(* CODESYS project 1102_xlh_stamp_rover_ddsm210_imu_client.project
   Author: 3S - Smart Software Solutions GmbH
   Version: 1.0.0.0
   Description: Receives some incoming messages and echoes them with CAN-ID +1
   Title: CAN Bus API Example
   Company: 3S - Smart Software Solutions GmbH

Project tree, tasks and I/O mapping:
  xLH_base : CODESYS Control for Raspberry Pi 64 SL, CODESYS, order no. 2302000009, version 4.20.0.0
    application app
      libraries: Standard, 3.5.22.0 (System); Util, 3.5.22.0 (System); VisuDialogs, * (System); Memory, * (3S - Smart Software Solutions GmbH); CmpBitmapPool, * (System); CAN API, 1.0.0.4 (CODESYS)
      task MAIN_TASK (cyclic, interval 5 ms, priority 0) calls MAIN
      program MAIN [ST]
    SoftMotion General Axis Pool
    GPIOs_A_B : GPIOs B+/Pi2, CODESYS, version 4.20.0.0
        unmapped channels: digital inputs (GPIO0..GPIO31), digital outputs (GPIO0..GPIO31)
    Onewire
    Camera device
      <Leer>
    SPI
    I²C
    CANbus : CANbus, CODESYS, version 4.3.0.0
        settings: Baudrate = 1000 kbit/s
      xlh_ddsm210_ultrasonic : CANopen Device, CODESYS, version 4.3.0.0
          settings: Vendor Name = 'xemax ag'; Product Name = 'xlh_ddsm210_imu'; OD_ObjectCount = 16#001D; Objects.Objects = (wIndex := 16#1000, bySubCnt := 16#1); Objects.Objects = (wIndex := 16#1001, bySubCnt := 16#1); Objects.Objects = (wIndex := 16#1003, bySubCnt := 16#04); Objects.Objects = (wIndex := 16#1005, bySubCnt := 16#1); Objects.Objects = (wIndex := 16#1006, bySubCnt := 16#1); Objects.Objects = (wIndex := 16#100C, bySubCnt := 16#1); Objects.Objects = (wIndex := 16#100D, bySubCnt := 16#1); Objects.Objects = (wIndex := 16#1016, bySubCnt := 16#02); Objects.Objects = (wIndex := 16#1018, bySubCnt := 16#04); Objects.Objects = (wIndex := 16#1200, bySubCnt := 16#03); Objects.Objects = (wIndex := 16#1400, bySubCnt := 16#03); Objects.Objects = (wIndex := 16#1600, bySubCnt := 16#05); Objects.Objects = (wIndex := 16#1800, bySubCnt := 16#06); Objects.Objects = (wIndex := 16#1801, bySubCnt := 16#06); Objects.Objects = (wIndex := 16#1802, bySubCnt := 16#06); Objects.Objects = (wIndex := 16#1A00, bySubCnt := 16#05); Objects.Objects = (wIndex := 16#1A01, bySubCnt := 16#03); Objects.Objects = (wIndex := 16#1A02, bySubCnt := 16#04); Objects.Objects = (wIndex := 16#3000, bySubCnt := 16#02); Objects.Objects = (wIndex := 16#3001, bySubCnt := 16#02); Objects.Objects = (wIndex := 16#3002, bySubCnt := 16#02); Objects.Objects = (wIndex := 16#3003, bySubCnt := 16#02); Objects.Objects = (wIndex := 16#3800, bySubCnt := 16#02); Objects.Objects = (wIndex := 16#3801, bySubCnt := 16#02); Objects.Objects = (wIndex := 16#3802, bySubCnt := 16#02); Objects.Objects = (wIndex := 16#3803, bySubCnt := 16#02); Objects.Objects = (wIndex := 16#3804, bySubCnt := 16#02); Objects.Objects = (wIndex := 16#3805, bySubCnt := 16#02); Objects.Objects = (wIndex := 16#3806, bySubCnt := 16#04); SubObjects.SubObjects = (eObjProperties := 16#0001, eDataType := 16#07, udiSize := 16#00000004, xwData := 0, xwDefault := 0, bySubIdx := 16#00); SubObjects.SubObjects = (eObjProperties := 16#0001, eDataType := 16#05, udiSize := 16#00000001, xwData := 0, xwDefault := 0, bySubIdx := 16#00); SubObjects.SubObjects = (eObjProperties := 16#0003, eDataType := 16#05, udiSize := 16#00000001, xwData := 0, xwDefault := 0, bySubIdx := 16#00); SubObjects.SubObjects = (eObjProperties := 16#0001, eDataType := 16#07, udiSize := 16#00000004, xwData := 0, xwDefault := 0, bySubIdx := 16#01); SubObjects.SubObjects = (eObjProperties := 16#0001, eDataType := 16#07, udiSize := 16#00000004, xwData := 0, xwDefault := 0, bySubIdx := 16#02); SubObjects.SubObjects = (eObjProperties := 16#0001, eDataType := 16#07, udiSize := 16#00000004, xwData := 0, xwDefault := 0, bySubIdx := 16#03); SubObjects.SubObjects = (eObjProperties := 16#0003, eDataType := 16#07, udiSize := 16#00000004, xwData := 0, xwDefault := 0, bySubIdx := 16#00); SubObjects.SubObjects = (eObjProperties := 16#0003, eDataType := 16#05, udiSize := 16#00000001, xwData := 0, xwDefault := 3, bySubIdx := 16#00);
            SubObjects.SubObjects = (eObjProperties := 16#0001, eDataType := 16#05, udiSize := 16#00000001, xwData := 0, xwDefault := 1, bySubIdx := 16#00); SubObjects.SubObjects = (eObjProperties := 16#0003, eDataType := 16#07, udiSize := 16#00000004, xwData := 0, xwDefault := 0, bySubIdx := 16#01); SubObjects.SubObjects = (eObjProperties := 16#0001, eDataType := 16#05, udiSize := 16#00000001, xwData := 0, xwDefault := 3, bySubIdx := 16#00); SubObjects.SubObjects = (eObjProperties := 16#0001, eDataType := 16#07, udiSize := 16#00000004, xwData := 0, xwDefault := 1, bySubIdx := 16#03); SubObjects.SubObjects = (eObjProperties := 16#0001, eDataType := 16#05, udiSize := 16#00000001, xwData := 0, xwDefault := 2, bySubIdx := 16#00); SubObjects.SubObjects = (eObjProperties := 16#0001, eDataType := 16#05, udiSize := 16#00000001, xwData := 0, xwDefault := 2, bySubIdx := 16#00); SubObjects.SubObjects = (eObjProperties := 16#0001, eDataType := 16#05, udiSize := 16#00000001, xwData := 0, xwDefault := 4, bySubIdx := 16#00); SubObjects.SubObjects = (eObjProperties := 16#0001, eDataType := 16#05, udiSize := 16#00000001, xwData := 0, xwDefault := 5, bySubIdx := 16#00); SubObjects.SubObjects = (eObjProperties := 16#0003, eDataType := 16#06, udiSize := 16#00000002, xwData := 0, xwDefault := 0, bySubIdx := 16#03); SubObjects.SubObjects = (eObjProperties := 16#0003, eDataType := 16#05, udiSize := 16#00000001, xwData := 0, xwDefault := 0, bySubIdx := 16#04); SubObjects.SubObjects = (eObjProperties := 16#0003, eDataType := 16#06, udiSize := 16#00000002, xwData := 0, xwDefault := 0, bySubIdx := 16#05); SubObjects.SubObjects = (eObjProperties := 16#0001, eDataType := 16#05, udiSize := 16#00000001, xwData := 0, xwDefault := 5, bySubIdx := 16#00); SubObjects.SubObjects = (eObjProperties := 16#0003, eDataType := 16#06, udiSize := 16#00000002, xwData := 0, xwDefault := 0, bySubIdx := 16#03); SubObjects.SubObjects = (eObjProperties := 16#0003, eDataType := 16#05, udiSize := 16#00000001, xwData := 0, xwDefault := 0, bySubIdx := 16#04); SubObjects.SubObjects = (eObjProperties := 16#0003, eDataType := 16#06, udiSize := 16#00000002, xwData := 0, xwDefault := 0, bySubIdx := 16#05); SubObjects.SubObjects = (eObjProperties := 16#0001, eDataType := 16#05, udiSize := 16#00000001, xwData := 0, xwDefault := 5, bySubIdx := 16#00); SubObjects.SubObjects = (eObjProperties := 16#0003, eDataType := 16#06, udiSize := 16#00000002, xwData := 0, xwDefault := 0, bySubIdx := 16#03); SubObjects.SubObjects = (eObjProperties := 16#0003, eDataType := 16#05, udiSize := 16#00000001, xwData := 0, xwDefault := 0, bySubIdx := 16#04); SubObjects.SubObjects = (eObjProperties := 16#0003, eDataType := 16#06, udiSize := 16#00000002, xwData := 0, xwDefault := 0, bySubIdx := 16#05); SubObjects.SubObjects = (eObjProperties := 16#0001, eDataType := 16#05, udiSize := 16#00000001, xwData := 0, xwDefault := 4, bySubIdx := 16#00); SubObjects.SubObjects = (eObjProperties := 16#0001, eDataType := 16#05, udiSize := 16#00000001, xwData := 0, xwDefault := 2, bySubIdx := 16#00); SubObjects.SubObjects = (eObjProperties := 16#0001, eDataType := 16#05, udiSize := 16#00000001, xwData := 0, xwDefault := 3, bySubIdx := 16#00); SubObjects.SubObjects = (eObjProperties := 16#0001, eDataType := 16#05, udiSize := 16#00000001, xwData := 0, xwDefault := 1, bySubIdx := 16#00); SubObjects.SubObjects = (eObjProperties := 16#0003, eDataType := 16#03, udiSize := 16#00000002, xwData := 0, xwDefault := 0, bySubIdx := 16#01); SubObjects.SubObjects = (eObjProperties := 16#0001, eDataType := 16#05, udiSize := 16#00000001, xwData := 0, xwDefault := 1, bySubIdx := 16#00); SubObjects.SubObjects = (eObjProperties := 16#0003, eDataType := 16#05, udiSize := 16#00000001, xwData := 0, xwDefault := 0, bySubIdx := 16#01); SubObjects.SubObjects = (eObjProperties := 16#0001, eDataType := 16#05, udiSize := 16#00000001, xwData := 0, xwDefault := 1, bySubIdx := 16#00); SubObjects.SubObjects = (eObjProperties := 16#0003, eDataType := 16#03, udiSize := 16#00000002, xwData := 0, xwDefault := 0, bySubIdx := 16#01); SubObjects.SubObjects = (eObjProperties := 16#0001, eDataType := 16#05, udiSize := 16#00000001, xwData := 0, xwDefault := 1, bySubIdx := 16#00); SubObjects.SubObjects = (eObjProperties := 16#0003, eDataType := 16#05, udiSize := 16#00000001, xwData := 0, xwDefault := 0, bySubIdx := 16#01); SubObjects.SubObjects = (eObjProperties := 16#0001, eDataType := 16#05, udiSize := 16#00000001, xwData := 0, xwDefault := 1, bySubIdx := 16#00); SubObjects.SubObjects = (eObjProperties := 16#0001, eDataType := 16#03, udiSize := 16#00000002, xwData := 0, xwDefault := 0, bySubIdx := 16#01); SubObjects.SubObjects = (eObjProperties := 16#0001, eDataType := 16#05, udiSize := 16#00000001, xwData := 0, xwDefault := 1, bySubIdx := 16#00); SubObjects.SubObjects = (eObjProperties := 16#0001, eDataType := 16#03, udiSize := 16#00000002, xwData := 0, xwDefault := 0, bySubIdx := 16#01); SubObjects.SubObjects = (eObjProperties := 16#0001, eDataType := 16#05, udiSize := 16#00000001, xwData := 0, xwDefault := 1, bySubIdx := 16#00); SubObjects.SubObjects = (eObjProperties := 16#0001, eDataType := 16#05, udiSize := 16#00000001, xwData := 0, xwDefault := 0, bySubIdx := 16#01); SubObjects.SubObjects = (eObjProperties := 16#0001, eDataType := 16#05, udiSize := 16#00000001, xwData := 0, xwDefault := 1, bySubIdx := 16#00); SubObjects.SubObjects = (eObjProperties := 16#0001, eDataType := 16#05, udiSize := 16#00000001, xwData := 0, xwDefault := 0, bySubIdx := 16#01); SubObjects.SubObjects = (eObjProperties := 16#0001, eDataType := 16#05, udiSize := 16#00000001, xwData := 0, xwDefault := 1, bySubIdx := 16#00); SubObjects.SubObjects = (eObjProperties := 16#0001, eDataType := 16#04, udiSize := 16#00000004, xwData := 0, xwDefault := 0, bySubIdx := 16#01);
            SubObjects.SubObjects = (eObjProperties := 16#0001, eDataType := 16#05, udiSize := 16#00000001, xwData := 0, xwDefault := 1, bySubIdx := 16#00); SubObjects.SubObjects = (eObjProperties := 16#0001, eDataType := 16#06, udiSize := 16#00000002, xwData := 0, xwDefault := 0, bySubIdx := 16#01); SubObjects.SubObjects = (eObjProperties := 16#0001, eDataType := 16#05, udiSize := 16#00000001, xwData := 0, xwDefault := 3, bySubIdx := 16#00); SubObjects.SubObjects = (eObjProperties := 16#0001, eDataType := 16#03, udiSize := 16#00000002, xwData := 0, xwDefault := 0, bySubIdx := 16#01); SubObjects.SubObjects = (eObjProperties := 16#0001, eDataType := 16#03, udiSize := 16#00000002, xwData := 0, xwDefault := 0, bySubIdx := 16#02); SubObjects.SubObjects = (eObjProperties := 16#0001, eDataType := 16#03, udiSize := 16#00000002, xwData := 0, xwDefault := 0, bySubIdx := 16#03); ObjectsOfflineInfo.Predefined Error Field.Index = 16#00001003; ObjectsOfflineInfo.Predefined Error Field.ObjectOwner = 16#00; ObjectsOfflineInfo.Predefined Error Field.ObjectType = 16#00000008; ObjectsOfflineInfo.Predefined Error Field.ObjectFlags = 16#00000000; ObjectsOfflineInfo.Consumer Heartbeat Time.Index = 16#00001016; ObjectsOfflineInfo.Consumer Heartbeat Time.ObjectOwner = 16#00; ObjectsOfflineInfo.Consumer Heartbeat Time.ObjectType = 16#00000008; ObjectsOfflineInfo.Consumer Heartbeat Time.ObjectFlags = 16#00000000; ObjectsOfflineInfo.Identity Object.Index = 16#00001018; ObjectsOfflineInfo.Identity Object.ObjectOwner = 16#00; ObjectsOfflineInfo.Identity Object.ObjectType = 16#00000009; ObjectsOfflineInfo.Identity Object.ObjectFlags = 16#00000000; ObjectsOfflineInfo.ServerSdoParameter.Index = 16#00001200; ObjectsOfflineInfo.ServerSdoParameter.ObjectOwner = 16#00; ObjectsOfflineInfo.ServerSdoParameter.ObjectType = 16#00000009; ObjectsOfflineInfo.ServerSdoParameter.ObjectFlags = 16#00000000; ObjectsOfflineInfo.RPDO communication parameter.Index = 16#00001400; ObjectsOfflineInfo.RPDO communication parameter.ObjectOwner = 16#03; ObjectsOfflineInfo.RPDO communication parameter.ObjectType = 16#00000009; ObjectsOfflineInfo.RPDO communication parameter.ObjectFlags = 16#00000000; ObjectsOfflineInfo.RPDO mapping parameter.Index = 16#00001600; ObjectsOfflineInfo.RPDO mapping parameter.ObjectOwner = 16#03; ObjectsOfflineInfo.RPDO mapping parameter.ObjectType = 16#00000009; ObjectsOfflineInfo.RPDO mapping parameter.ObjectFlags = 16#00000000; ObjectsOfflineInfo.TPDO communication parameter.Index = 16#00001800; ObjectsOfflineInfo.TPDO communication parameter.ObjectOwner = 16#03; ObjectsOfflineInfo.TPDO communication parameter.ObjectType = 16#00000009; ObjectsOfflineInfo.TPDO communication parameter.ObjectFlags = 16#00000000; ObjectsOfflineInfo.TPDO communication parameter.Index = 16#00001801; ObjectsOfflineInfo.TPDO communication parameter.ObjectOwner = 16#03; ObjectsOfflineInfo.TPDO communication parameter.ObjectType = 16#00000009; ObjectsOfflineInfo.TPDO communication parameter.ObjectFlags = 16#00000000; ObjectsOfflineInfo.TPDO communication parameter.Index = 16#00001802; ObjectsOfflineInfo.TPDO communication parameter.ObjectOwner = 16#03;
            ObjectsOfflineInfo.TPDO communication parameter.ObjectType = 16#00000009; ObjectsOfflineInfo.TPDO communication parameter.ObjectFlags = 16#00000000; ObjectsOfflineInfo.TPDO mapping parameter.Index = 16#00001A00; ObjectsOfflineInfo.TPDO mapping parameter.ObjectOwner = 16#03; ObjectsOfflineInfo.TPDO mapping parameter.ObjectType = 16#00000009; ObjectsOfflineInfo.TPDO mapping parameter.ObjectFlags = 16#00000000; ObjectsOfflineInfo.TPDO mapping parameter.Index = 16#00001A01; ObjectsOfflineInfo.TPDO mapping parameter.ObjectOwner = 16#03; ObjectsOfflineInfo.TPDO mapping parameter.ObjectType = 16#00000009; ObjectsOfflineInfo.TPDO mapping parameter.ObjectFlags = 16#00000000; ObjectsOfflineInfo.TPDO mapping parameter.Index = 16#00001A02; ObjectsOfflineInfo.TPDO mapping parameter.ObjectOwner = 16#03; ObjectsOfflineInfo.TPDO mapping parameter.ObjectType = 16#00000009; ObjectsOfflineInfo.TPDO mapping parameter.ObjectFlags = 16#00000000; ObjectsOfflineInfo.set_speed.Index = 16#00003000; ObjectsOfflineInfo.set_speed.ObjectOwner = 16#03; ObjectsOfflineInfo.set_speed.ObjectType = 16#00000008; ObjectsOfflineInfo.set_speed.ObjectFlags = 16#00000000; ObjectsOfflineInfo.set_acc_time.Index = 16#00003001; ObjectsOfflineInfo.set_acc_time.ObjectOwner = 16#03; ObjectsOfflineInfo.set_acc_time.ObjectType = 16#00000008; ObjectsOfflineInfo.set_acc_time.ObjectFlags = 16#00000000; ObjectsOfflineInfo.set_current_limit.Index = 16#00003002; ObjectsOfflineInfo.set_current_limit.ObjectOwner = 16#03; ObjectsOfflineInfo.set_current_limit.ObjectType = 16#00000008; ObjectsOfflineInfo.set_current_limit.ObjectFlags = 16#00000000; ObjectsOfflineInfo.set_cmd.Index = 16#00003003; ObjectsOfflineInfo.set_cmd.ObjectOwner = 16#03; ObjectsOfflineInfo.set_cmd.ObjectType = 16#00000008; ObjectsOfflineInfo.set_cmd.ObjectFlags = 16#00000000; ObjectsOfflineInfo.speed.Index = 16#00003800; ObjectsOfflineInfo.speed.ObjectOwner = 16#03; ObjectsOfflineInfo.speed.ObjectType = 16#00000008; ObjectsOfflineInfo.speed.ObjectFlags = 16#00000000; ObjectsOfflineInfo.current.Index = 16#00003801; ObjectsOfflineInfo.current.ObjectOwner = 16#03; ObjectsOfflineInfo.current.ObjectType = 16#00000008; ObjectsOfflineInfo.current.ObjectFlags = 16#00000000; ObjectsOfflineInfo.acc_time.Index = 16#00003802; ObjectsOfflineInfo.acc_time.ObjectOwner = 16#03;
            ObjectsOfflineInfo.acc_time.ObjectType = 16#00000008; ObjectsOfflineInfo.acc_time.ObjectFlags = 16#00000000; ObjectsOfflineInfo.temperature.Index = 16#00003803; ObjectsOfflineInfo.temperature.ObjectOwner = 16#03; ObjectsOfflineInfo.temperature.ObjectType = 16#00000008; ObjectsOfflineInfo.temperature.ObjectFlags = 16#00000000; ObjectsOfflineInfo.position.Index = 16#00003804; ObjectsOfflineInfo.position.ObjectOwner = 16#03; ObjectsOfflineInfo.position.ObjectType = 16#00000008; ObjectsOfflineInfo.position.ObjectFlags = 16#00000000; ObjectsOfflineInfo.error_code.Index = 16#00003805; ObjectsOfflineInfo.error_code.ObjectOwner = 16#03; ObjectsOfflineInfo.error_code.ObjectType = 16#00000008; ObjectsOfflineInfo.error_code.ObjectFlags = 16#00000000; ObjectsOfflineInfo.imu.Index = 16#00003806; ObjectsOfflineInfo.imu.ObjectOwner = 16#03; ObjectsOfflineInfo.imu.ObjectType = 16#00000008; ObjectsOfflineInfo.imu.ObjectFlags = 16#00000000; SubObjectsOfflineInfo.Device Type.Index = 16#00001000; SubObjectsOfflineInfo.Device Type.SubIndex = 16#00; SubObjectsOfflineInfo.Device Type.PDOMapping = FALSE; SubObjectsOfflineInfo.Device Type.ObjectOwner = 16#00; SubObjectsOfflineInfo.Device Type.ObjectType = 16#00000007; SubObjectsOfflineInfo.Device Type.MinValue = ''; SubObjectsOfflineInfo.Device Type.MaxValue = ''; SubObjectsOfflineInfo.Device Type.AccessType = 'ro'; SubObjectsOfflineInfo.Device Type.IEC Variable = ''; SubObjectsOfflineInfo.Device Type.DefaultValue = '0x0'; SubObjectsOfflineInfo.Device Type.ObjectFlags = 16#00000000; SubObjectsOfflineInfo.Error Register.Index = 16#00001001; SubObjectsOfflineInfo.Error Register.SubIndex = 16#00; SubObjectsOfflineInfo.Error Register.PDOMapping = FALSE; SubObjectsOfflineInfo.Error Register.ObjectOwner = 16#00; SubObjectsOfflineInfo.Error Register.ObjectType = 16#00000007; SubObjectsOfflineInfo.Error Register.MinValue = ''; SubObjectsOfflineInfo.Error Register.MaxValue = ''; SubObjectsOfflineInfo.Error Register.AccessType = 'ro'; SubObjectsOfflineInfo.Error Register.IEC Variable = ''; SubObjectsOfflineInfo.Error Register.DefaultValue = '0x0'; SubObjectsOfflineInfo.Error Register.ObjectFlags = 16#00000000;
            SubObjectsOfflineInfo.Number of Errors.Index = 16#00001003; SubObjectsOfflineInfo.Number of Errors.SubIndex = 16#00; SubObjectsOfflineInfo.Number of Errors.PDOMapping = FALSE; SubObjectsOfflineInfo.Number of Errors.ObjectOwner = 16#00; SubObjectsOfflineInfo.Number of Errors.ObjectType = 16#00000007; SubObjectsOfflineInfo.Number of Errors.MinValue = ''; SubObjectsOfflineInfo.Number of Errors.MaxValue = ''; SubObjectsOfflineInfo.Number of Errors.AccessType = 'rw'; SubObjectsOfflineInfo.Number of Errors.IEC Variable = ''; SubObjectsOfflineInfo.Number of Errors.DefaultValue = '0'; SubObjectsOfflineInfo.Number of Errors.ObjectFlags = 16#00000000; SubObjectsOfflineInfo.Standard Error Field.Index = 16#00001003; SubObjectsOfflineInfo.Standard Error Field.SubIndex = 16#01; SubObjectsOfflineInfo.Standard Error Field.PDOMapping = FALSE; SubObjectsOfflineInfo.Standard Error Field.ObjectOwner = 16#00; SubObjectsOfflineInfo.Standard Error Field.ObjectType = 16#00000007; SubObjectsOfflineInfo.Standard Error Field.MinValue = ''; SubObjectsOfflineInfo.Standard Error Field.MaxValue = ''; SubObjectsOfflineInfo.Standard Error Field.AccessType = 'ro'; SubObjectsOfflineInfo.Standard Error Field.IEC Variable = ''; SubObjectsOfflineInfo.Standard Error Field.DefaultValue = ''; SubObjectsOfflineInfo.Standard Error Field.ObjectFlags = 16#00000000; SubObjectsOfflineInfo.Standard Error Field 2.Index = 16#00001003; SubObjectsOfflineInfo.Standard Error Field 2.SubIndex = 16#02; SubObjectsOfflineInfo.Standard Error Field 2.PDOMapping = FALSE; SubObjectsOfflineInfo.Standard Error Field 2.ObjectOwner = 16#00; SubObjectsOfflineInfo.Standard Error Field 2.ObjectType = 16#00000007; SubObjectsOfflineInfo.Standard Error Field 2.MinValue = ''; SubObjectsOfflineInfo.Standard Error Field 2.MaxValue = ''; SubObjectsOfflineInfo.Standard Error Field 2.AccessType = 'ro'; SubObjectsOfflineInfo.Standard Error Field 2.IEC Variable = ''; SubObjectsOfflineInfo.Standard Error Field 2.DefaultValue = ''; SubObjectsOfflineInfo.Standard Error Field 2.ObjectFlags = 16#00000000; SubObjectsOfflineInfo.Standard Error Field 3.Index = 16#00001003; SubObjectsOfflineInfo.Standard Error Field 3.SubIndex = 16#03; SubObjectsOfflineInfo.Standard Error Field 3.PDOMapping = FALSE; SubObjectsOfflineInfo.Standard Error Field 3.ObjectOwner = 16#00; SubObjectsOfflineInfo.Standard Error Field 3.ObjectType = 16#00000007; SubObjectsOfflineInfo.Standard Error Field 3.MinValue = ''; SubObjectsOfflineInfo.Standard Error Field 3.MaxValue = '';
            SubObjectsOfflineInfo.Standard Error Field 3.AccessType = 'ro'; SubObjectsOfflineInfo.Standard Error Field 3.IEC Variable = ''; SubObjectsOfflineInfo.Standard Error Field 3.DefaultValue = ''; SubObjectsOfflineInfo.Standard Error Field 3.ObjectFlags = 16#00000000; SubObjectsOfflineInfo.Sync COB-ID.Index = 16#00001005; SubObjectsOfflineInfo.Sync COB-ID.SubIndex = 16#00; SubObjectsOfflineInfo.Sync COB-ID.PDOMapping = FALSE; SubObjectsOfflineInfo.Sync COB-ID.ObjectOwner = 16#00; SubObjectsOfflineInfo.Sync COB-ID.ObjectType = 16#00000007; SubObjectsOfflineInfo.Sync COB-ID.MinValue = ''; SubObjectsOfflineInfo.Sync COB-ID.MaxValue = ''; SubObjectsOfflineInfo.Sync COB-ID.AccessType = 'rw'; SubObjectsOfflineInfo.Sync COB-ID.IEC Variable = ''; SubObjectsOfflineInfo.Sync COB-ID.DefaultValue = '0x80'; SubObjectsOfflineInfo.Sync COB-ID.ObjectFlags = 16#00000000; SubObjectsOfflineInfo.Communication Cycle Period.Index = 16#00001006; SubObjectsOfflineInfo.Communication Cycle Period.SubIndex = 16#00; SubObjectsOfflineInfo.Communication Cycle Period.PDOMapping = FALSE; SubObjectsOfflineInfo.Communication Cycle Period.ObjectOwner = 16#00; SubObjectsOfflineInfo.Communication Cycle Period.ObjectType = 16#00000007; SubObjectsOfflineInfo.Communication Cycle Period.MinValue = ''; SubObjectsOfflineInfo.Communication Cycle Period.MaxValue = ''; SubObjectsOfflineInfo.Communication Cycle Period.AccessType = 'rw'; SubObjectsOfflineInfo.Communication Cycle Period.IEC Variable = ''; SubObjectsOfflineInfo.Communication Cycle Period.DefaultValue = '0x0'; SubObjectsOfflineInfo.Communication Cycle Period.ObjectFlags = 16#00000000; SubObjectsOfflineInfo.Guard Time.Index = 16#0000100C; SubObjectsOfflineInfo.Guard Time.SubIndex = 16#00; SubObjectsOfflineInfo.Guard Time.PDOMapping = FALSE; SubObjectsOfflineInfo.Guard Time.ObjectOwner = 16#00; SubObjectsOfflineInfo.Guard Time.ObjectType = 16#00000007; SubObjectsOfflineInfo.Guard Time.MinValue = ''; SubObjectsOfflineInfo.Guard Time.MaxValue = ''; SubObjectsOfflineInfo.Guard Time.AccessType = 'rw'; SubObjectsOfflineInfo.Guard Time.IEC Variable = ''; SubObjectsOfflineInfo.Guard Time.DefaultValue = '200'; SubObjectsOfflineInfo.Guard Time.ObjectFlags = 16#00000000; SubObjectsOfflineInfo.Life Time Factor.Index = 16#0000100D; SubObjectsOfflineInfo.Life Time Factor.SubIndex = 16#00; SubObjectsOfflineInfo.Life Time Factor.PDOMapping = FALSE;
            SubObjectsOfflineInfo.Life Time Factor.ObjectOwner = 16#00; SubObjectsOfflineInfo.Life Time Factor.ObjectType = 16#00000007; SubObjectsOfflineInfo.Life Time Factor.MinValue = ''; SubObjectsOfflineInfo.Life Time Factor.MaxValue = ''; SubObjectsOfflineInfo.Life Time Factor.AccessType = 'rw'; SubObjectsOfflineInfo.Life Time Factor.IEC Variable = ''; SubObjectsOfflineInfo.Life Time Factor.DefaultValue = '3'; SubObjectsOfflineInfo.Life Time Factor.ObjectFlags = 16#00000000; SubObjectsOfflineInfo.Number of Entries.Index = 16#00001016; SubObjectsOfflineInfo.Number of Entries.SubIndex = 16#00; SubObjectsOfflineInfo.Number of Entries.PDOMapping = FALSE; SubObjectsOfflineInfo.Number of Entries.ObjectOwner = 16#00; SubObjectsOfflineInfo.Number of Entries.ObjectType = 16#00000007; SubObjectsOfflineInfo.Number of Entries.MinValue = ''; SubObjectsOfflineInfo.Number of Entries.MaxValue = ''; SubObjectsOfflineInfo.Number of Entries.AccessType = 'ro'; SubObjectsOfflineInfo.Number of Entries.IEC Variable = ''; SubObjectsOfflineInfo.Number of Entries.DefaultValue = '0x1'; SubObjectsOfflineInfo.Number of Entries.ObjectFlags = 16#00000000; SubObjectsOfflineInfo.Consumer Heartbeat Time.Index = 16#00001016; SubObjectsOfflineInfo.Consumer Heartbeat Time.SubIndex = 16#01; SubObjectsOfflineInfo.Consumer Heartbeat Time.PDOMapping = FALSE; SubObjectsOfflineInfo.Consumer Heartbeat Time.ObjectOwner = 16#00; SubObjectsOfflineInfo.Consumer Heartbeat Time.ObjectType = 16#00000007; SubObjectsOfflineInfo.Consumer Heartbeat Time.MinValue = ''; SubObjectsOfflineInfo.Consumer Heartbeat Time.MaxValue = ''; SubObjectsOfflineInfo.Consumer Heartbeat Time.AccessType = 'rw'; SubObjectsOfflineInfo.Consumer Heartbeat Time.IEC Variable = ''; SubObjectsOfflineInfo.Consumer Heartbeat Time.DefaultValue = '0x0'; SubObjectsOfflineInfo.Consumer Heartbeat Time.ObjectFlags = 16#00000000; SubObjectsOfflineInfo.Number of Entries.Index = 16#00001018; SubObjectsOfflineInfo.Number of Entries.SubIndex = 16#00; SubObjectsOfflineInfo.Number of Entries.PDOMapping = FALSE; SubObjectsOfflineInfo.Number of Entries.ObjectOwner = 16#00; SubObjectsOfflineInfo.Number of Entries.ObjectType = 16#00000007; SubObjectsOfflineInfo.Number of Entries.MinValue = '0x1'; SubObjectsOfflineInfo.Number of Entries.MaxValue = '0x3'; SubObjectsOfflineInfo.Number of Entries.AccessType = 'ro'; SubObjectsOfflineInfo.Number of Entries.IEC Variable = ''; SubObjectsOfflineInfo.Number of Entries.DefaultValue = '3';
            SubObjectsOfflineInfo.Number of Entries.ObjectFlags = 16#00000000; SubObjectsOfflineInfo.Vendor Id.Index = 16#00001018; SubObjectsOfflineInfo.Vendor Id.SubIndex = 16#01; SubObjectsOfflineInfo.Vendor Id.PDOMapping = FALSE; SubObjectsOfflineInfo.Vendor Id.ObjectOwner = 16#00; SubObjectsOfflineInfo.Vendor Id.ObjectType = 16#00000007; SubObjectsOfflineInfo.Vendor Id.MinValue = ''; SubObjectsOfflineInfo.Vendor Id.MaxValue = ''; SubObjectsOfflineInfo.Vendor Id.AccessType = 'ro'; SubObjectsOfflineInfo.Vendor Id.IEC Variable = ''; SubObjectsOfflineInfo.Vendor Id.DefaultValue = '801'; SubObjectsOfflineInfo.Vendor Id.ObjectFlags = 16#00000000; SubObjectsOfflineInfo.Product Code.Index = 16#00001018; SubObjectsOfflineInfo.Product Code.SubIndex = 16#02; SubObjectsOfflineInfo.Product Code.PDOMapping = FALSE; SubObjectsOfflineInfo.Product Code.ObjectOwner = 16#00; SubObjectsOfflineInfo.Product Code.ObjectType = 16#00000007; SubObjectsOfflineInfo.Product Code.MinValue = ''; SubObjectsOfflineInfo.Product Code.MaxValue = ''; SubObjectsOfflineInfo.Product Code.AccessType = 'ro'; SubObjectsOfflineInfo.Product Code.IEC Variable = ''; SubObjectsOfflineInfo.Product Code.DefaultValue = '1102'; SubObjectsOfflineInfo.Product Code.ObjectFlags = 16#00000000; SubObjectsOfflineInfo.Revision Number.Index = 16#00001018; SubObjectsOfflineInfo.Revision Number.SubIndex = 16#03; SubObjectsOfflineInfo.Revision Number.PDOMapping = FALSE; SubObjectsOfflineInfo.Revision Number.ObjectOwner = 16#00; SubObjectsOfflineInfo.Revision Number.ObjectType = 16#00000007; SubObjectsOfflineInfo.Revision Number.MinValue = ''; SubObjectsOfflineInfo.Revision Number.MaxValue = ''; SubObjectsOfflineInfo.Revision Number.AccessType = 'ro'; SubObjectsOfflineInfo.Revision Number.IEC Variable = ''; SubObjectsOfflineInfo.Revision Number.DefaultValue = '1'; SubObjectsOfflineInfo.Revision Number.ObjectFlags = 16#00000000; SubObjectsOfflineInfo.Number of Entries.Index = 16#00001200; SubObjectsOfflineInfo.Number of Entries.SubIndex = 16#00; SubObjectsOfflineInfo.Number of Entries.PDOMapping = FALSE; SubObjectsOfflineInfo.Number of Entries.ObjectOwner = 16#00; SubObjectsOfflineInfo.Number of Entries.ObjectType = 16#00000007; SubObjectsOfflineInfo.Number of Entries.MinValue = '0x2';
            SubObjectsOfflineInfo.Number of Entries.MaxValue = '0x2'; SubObjectsOfflineInfo.Number of Entries.AccessType = 'ro'; SubObjectsOfflineInfo.Number of Entries.IEC Variable = ''; SubObjectsOfflineInfo.Number of Entries.DefaultValue = '0x2'; SubObjectsOfflineInfo.Number of Entries.ObjectFlags = 16#00000000; SubObjectsOfflineInfo.COB-ID Client->Server.Index = 16#00001200; SubObjectsOfflineInfo.COB-ID Client->Server.SubIndex = 16#01; SubObjectsOfflineInfo.COB-ID Client->Server.PDOMapping = FALSE; SubObjectsOfflineInfo.COB-ID Client->Server.ObjectOwner = 16#00; SubObjectsOfflineInfo.COB-ID Client->Server.ObjectType = 16#00000007; SubObjectsOfflineInfo.COB-ID Client->Server.MinValue = ''; SubObjectsOfflineInfo.COB-ID Client->Server.MaxValue = ''; SubObjectsOfflineInfo.COB-ID Client->Server.AccessType = 'ro'; SubObjectsOfflineInfo.COB-ID Client->Server.IEC Variable = ''; SubObjectsOfflineInfo.COB-ID Client->Server.DefaultValue = '$$NodeId+0x600'; SubObjectsOfflineInfo.COB-ID Client->Server.ObjectFlags = 16#00000000; SubObjectsOfflineInfo.COB-ID Server->Client.Index = 16#00001200; SubObjectsOfflineInfo.COB-ID Server->Client.SubIndex = 16#02; SubObjectsOfflineInfo.COB-ID Server->Client.PDOMapping = FALSE; SubObjectsOfflineInfo.COB-ID Server->Client.ObjectOwner = 16#00; SubObjectsOfflineInfo.COB-ID Server->Client.ObjectType = 16#00000007; SubObjectsOfflineInfo.COB-ID Server->Client.MinValue = ''; SubObjectsOfflineInfo.COB-ID Server->Client.MaxValue = ''; SubObjectsOfflineInfo.COB-ID Server->Client.AccessType = 'ro'; SubObjectsOfflineInfo.COB-ID Server->Client.IEC Variable = ''; SubObjectsOfflineInfo.COB-ID Server->Client.DefaultValue = '$$NodeId+0x580'; SubObjectsOfflineInfo.COB-ID Server->Client.ObjectFlags = 16#00000000; SubObjectsOfflineInfo.Highest sub-index supported.Index = 16#00001400; SubObjectsOfflineInfo.Highest sub-index supported.SubIndex = 16#00; SubObjectsOfflineInfo.Highest sub-index supported.PDOMapping = FALSE; SubObjectsOfflineInfo.Highest sub-index supported.ObjectOwner = 16#03; SubObjectsOfflineInfo.Highest sub-index supported.ObjectType = 16#00000007; SubObjectsOfflineInfo.Highest sub-index supported.MinValue = '0x02'; SubObjectsOfflineInfo.Highest sub-index supported.MaxValue = '0x05'; SubObjectsOfflineInfo.Highest sub-index supported.AccessType = 'const'; SubObjectsOfflineInfo.Highest sub-index supported.IEC Variable = ''; SubObjectsOfflineInfo.Highest sub-index supported.DefaultValue = '0x2'; SubObjectsOfflineInfo.Highest sub-index supported.ObjectFlags = 16#00000000; SubObjectsOfflineInfo.COB-ID used by RPDO.Index = 16#00001400; SubObjectsOfflineInfo.COB-ID used by RPDO.SubIndex = 16#01;
            SubObjectsOfflineInfo.COB-ID used by RPDO.PDOMapping = FALSE; SubObjectsOfflineInfo.COB-ID used by RPDO.ObjectOwner = 16#03; SubObjectsOfflineInfo.COB-ID used by RPDO.ObjectType = 16#00000007; SubObjectsOfflineInfo.COB-ID used by RPDO.MinValue = '0x00000080'; SubObjectsOfflineInfo.COB-ID used by RPDO.MaxValue = '0xFFFFFFFF'; SubObjectsOfflineInfo.COB-ID used by RPDO.AccessType = 'rw'; SubObjectsOfflineInfo.COB-ID used by RPDO.IEC Variable = ''; SubObjectsOfflineInfo.COB-ID used by RPDO.DefaultValue = '$$NODEID+0x200'; SubObjectsOfflineInfo.COB-ID used by RPDO.ObjectFlags = 16#00000000; SubObjectsOfflineInfo.Transmission type.Index = 16#00001400; SubObjectsOfflineInfo.Transmission type.SubIndex = 16#02; SubObjectsOfflineInfo.Transmission type.PDOMapping = FALSE; SubObjectsOfflineInfo.Transmission type.ObjectOwner = 16#03; SubObjectsOfflineInfo.Transmission type.ObjectType = 16#00000007; SubObjectsOfflineInfo.Transmission type.MinValue = '0x00'; SubObjectsOfflineInfo.Transmission type.MaxValue = '0xFF'; SubObjectsOfflineInfo.Transmission type.AccessType = 'rw'; SubObjectsOfflineInfo.Transmission type.IEC Variable = ''; SubObjectsOfflineInfo.Transmission type.DefaultValue = '0xFF'; SubObjectsOfflineInfo.Transmission type.ObjectFlags = 16#00000000; SubObjectsOfflineInfo.Number of mapped application objects in PDO.Index = 16#00001600; SubObjectsOfflineInfo.Number of mapped application objects in PDO.SubIndex = 16#00; SubObjectsOfflineInfo.Number of mapped application objects in PDO.PDOMapping = FALSE; SubObjectsOfflineInfo.Number of mapped application objects in PDO.ObjectOwner = 16#03; SubObjectsOfflineInfo.Number of mapped application objects in PDO.ObjectType = 16#00000007; SubObjectsOfflineInfo.Number of mapped application objects in PDO.MinValue = '0x00'; SubObjectsOfflineInfo.Number of mapped application objects in PDO.MaxValue = '0xFF'; SubObjectsOfflineInfo.Number of mapped application objects in PDO.AccessType = 'const'; SubObjectsOfflineInfo.Number of mapped application objects in PDO.IEC Variable = ''; SubObjectsOfflineInfo.Number of mapped application objects in PDO.DefaultValue = '0x04'; SubObjectsOfflineInfo.Number of mapped application objects in PDO.ObjectFlags = 16#00000000; SubObjectsOfflineInfo.Mapping Entry.Index = 16#00001600; SubObjectsOfflineInfo.Mapping Entry.SubIndex = 16#01; SubObjectsOfflineInfo.Mapping Entry.PDOMapping = FALSE; SubObjectsOfflineInfo.Mapping Entry.ObjectOwner = 16#03; SubObjectsOfflineInfo.Mapping Entry.ObjectType = 16#00000007; SubObjectsOfflineInfo.Mapping Entry.MinValue = '0x0'; SubObjectsOfflineInfo.Mapping Entry.MaxValue = '0xFFFFFFFF'; SubObjectsOfflineInfo.Mapping Entry.AccessType = 'const'; SubObjectsOfflineInfo.Mapping Entry.IEC Variable = '';
            SubObjectsOfflineInfo.Mapping Entry.DefaultValue = '0x30000110'; SubObjectsOfflineInfo.Mapping Entry.ObjectFlags = 16#00000000; SubObjectsOfflineInfo.Mapping Entry.Index = 16#00001600; SubObjectsOfflineInfo.Mapping Entry.SubIndex = 16#02; SubObjectsOfflineInfo.Mapping Entry.PDOMapping = FALSE; SubObjectsOfflineInfo.Mapping Entry.ObjectOwner = 16#03; SubObjectsOfflineInfo.Mapping Entry.ObjectType = 16#00000007; SubObjectsOfflineInfo.Mapping Entry.MinValue = '0x0'; SubObjectsOfflineInfo.Mapping Entry.MaxValue = '0xFFFFFFFF'; SubObjectsOfflineInfo.Mapping Entry.AccessType = 'const'; SubObjectsOfflineInfo.Mapping Entry.IEC Variable = ''; SubObjectsOfflineInfo.Mapping Entry.DefaultValue = '0x30020110'; SubObjectsOfflineInfo.Mapping Entry.ObjectFlags = 16#00000000; SubObjectsOfflineInfo.Mapping Entry.Index = 16#00001600; SubObjectsOfflineInfo.Mapping Entry.SubIndex = 16#03; SubObjectsOfflineInfo.Mapping Entry.PDOMapping = FALSE; SubObjectsOfflineInfo.Mapping Entry.ObjectOwner = 16#03; SubObjectsOfflineInfo.Mapping Entry.ObjectType = 16#00000007; SubObjectsOfflineInfo.Mapping Entry.MinValue = '0x0'; SubObjectsOfflineInfo.Mapping Entry.MaxValue = '0xFFFFFFFF'; SubObjectsOfflineInfo.Mapping Entry.AccessType = 'const'; SubObjectsOfflineInfo.Mapping Entry.IEC Variable = ''; SubObjectsOfflineInfo.Mapping Entry.DefaultValue = '0x30010108'; SubObjectsOfflineInfo.Mapping Entry.ObjectFlags = 16#00000000; SubObjectsOfflineInfo.Mapping Entry.Index = 16#00001600; SubObjectsOfflineInfo.Mapping Entry.SubIndex = 16#04; SubObjectsOfflineInfo.Mapping Entry.PDOMapping = FALSE; SubObjectsOfflineInfo.Mapping Entry.ObjectOwner = 16#03; SubObjectsOfflineInfo.Mapping Entry.ObjectType = 16#00000007; SubObjectsOfflineInfo.Mapping Entry.MinValue = '0x0'; SubObjectsOfflineInfo.Mapping Entry.MaxValue = '0xFFFFFFFF'; SubObjectsOfflineInfo.Mapping Entry.AccessType = 'const'; SubObjectsOfflineInfo.Mapping Entry.IEC Variable = ''; SubObjectsOfflineInfo.Mapping Entry.DefaultValue = '0x30030108'; SubObjectsOfflineInfo.Mapping Entry.ObjectFlags = 16#00000000; SubObjectsOfflineInfo.Highest sub-index supported.Index = 16#00001800; SubObjectsOfflineInfo.Highest sub-index supported.SubIndex = 16#00; SubObjectsOfflineInfo.Highest sub-index supported.PDOMapping = FALSE; SubObjectsOfflineInfo.Highest sub-index supported.ObjectOwner = 16#03; SubObjectsOfflineInfo.Highest sub-index supported.ObjectType = 16#00000007;
            SubObjectsOfflineInfo.Highest sub-index supported.MinValue = '0x02'; SubObjectsOfflineInfo.Highest sub-index supported.MaxValue = '0x06'; SubObjectsOfflineInfo.Highest sub-index supported.AccessType = 'const'; SubObjectsOfflineInfo.Highest sub-index supported.IEC Variable = ''; SubObjectsOfflineInfo.Highest sub-index supported.DefaultValue = '0x5'; SubObjectsOfflineInfo.Highest sub-index supported.ObjectFlags = 16#00000000; SubObjectsOfflineInfo.COB-ID used by TPDO.Index = 16#00001800; SubObjectsOfflineInfo.COB-ID used by TPDO.SubIndex = 16#01; SubObjectsOfflineInfo.COB-ID used by TPDO.PDOMapping = FALSE; SubObjectsOfflineInfo.COB-ID used by TPDO.ObjectOwner = 16#03; SubObjectsOfflineInfo.COB-ID used by TPDO.ObjectType = 16#00000007; SubObjectsOfflineInfo.COB-ID used by TPDO.MinValue = '0x00000080'; SubObjectsOfflineInfo.COB-ID used by TPDO.MaxValue = '0xFFFFFFFF'; SubObjectsOfflineInfo.COB-ID used by TPDO.AccessType = 'rw'; SubObjectsOfflineInfo.COB-ID used by TPDO.IEC Variable = ''; SubObjectsOfflineInfo.COB-ID used by TPDO.DefaultValue = '$$NODEID+0x180'; SubObjectsOfflineInfo.COB-ID used by TPDO.ObjectFlags = 16#00000000; SubObjectsOfflineInfo.Transmission type.Index = 16#00001800; SubObjectsOfflineInfo.Transmission type.SubIndex = 16#02; SubObjectsOfflineInfo.Transmission type.PDOMapping = FALSE; SubObjectsOfflineInfo.Transmission type.ObjectOwner = 16#03; SubObjectsOfflineInfo.Transmission type.ObjectType = 16#00000007; SubObjectsOfflineInfo.Transmission type.MinValue = '0x00'; SubObjectsOfflineInfo.Transmission type.MaxValue = '0xFF'; SubObjectsOfflineInfo.Transmission type.AccessType = 'rw'; SubObjectsOfflineInfo.Transmission type.IEC Variable = ''; SubObjectsOfflineInfo.Transmission type.DefaultValue = '0xFF'; SubObjectsOfflineInfo.Transmission type.ObjectFlags = 16#00000000; SubObjectsOfflineInfo.Inhibit time.Index = 16#00001800; SubObjectsOfflineInfo.Inhibit time.SubIndex = 16#03; SubObjectsOfflineInfo.Inhibit time.PDOMapping = FALSE; SubObjectsOfflineInfo.Inhibit time.ObjectOwner = 16#03; SubObjectsOfflineInfo.Inhibit time.ObjectType = 16#00000007; SubObjectsOfflineInfo.Inhibit time.MinValue = ''; SubObjectsOfflineInfo.Inhibit time.MaxValue = ''; SubObjectsOfflineInfo.Inhibit time.AccessType = 'rw'; SubObjectsOfflineInfo.Inhibit time.IEC Variable = ''; SubObjectsOfflineInfo.Inhibit time.DefaultValue = '0x0'; SubObjectsOfflineInfo.Inhibit time.ObjectFlags = 16#00000000; SubObjectsOfflineInfo.compatibility entry.Index = 16#00001800;
            SubObjectsOfflineInfo.compatibility entry.SubIndex = 16#04; SubObjectsOfflineInfo.compatibility entry.PDOMapping = FALSE; SubObjectsOfflineInfo.compatibility entry.ObjectOwner = 16#03; SubObjectsOfflineInfo.compatibility entry.ObjectType = 16#00000007; SubObjectsOfflineInfo.compatibility entry.MinValue = ''; SubObjectsOfflineInfo.compatibility entry.MaxValue = ''; SubObjectsOfflineInfo.compatibility entry.AccessType = 'rw'; SubObjectsOfflineInfo.compatibility entry.IEC Variable = ''; SubObjectsOfflineInfo.compatibility entry.DefaultValue = '0x0'; SubObjectsOfflineInfo.compatibility entry.ObjectFlags = 16#00000000; SubObjectsOfflineInfo.Event timer.Index = 16#00001800; SubObjectsOfflineInfo.Event timer.SubIndex = 16#05; SubObjectsOfflineInfo.Event timer.PDOMapping = FALSE; SubObjectsOfflineInfo.Event timer.ObjectOwner = 16#03; SubObjectsOfflineInfo.Event timer.ObjectType = 16#00000007; SubObjectsOfflineInfo.Event timer.MinValue = ''; SubObjectsOfflineInfo.Event timer.MaxValue = ''; SubObjectsOfflineInfo.Event timer.AccessType = 'rw'; SubObjectsOfflineInfo.Event timer.IEC Variable = ''; SubObjectsOfflineInfo.Event timer.DefaultValue = '0x0'; SubObjectsOfflineInfo.Event timer.ObjectFlags = 16#00000000; SubObjectsOfflineInfo.Highest sub-index supported.Index = 16#00001801; SubObjectsOfflineInfo.Highest sub-index supported.SubIndex = 16#00; SubObjectsOfflineInfo.Highest sub-index supported.PDOMapping = FALSE; SubObjectsOfflineInfo.Highest sub-index supported.ObjectOwner = 16#03; SubObjectsOfflineInfo.Highest sub-index supported.ObjectType = 16#00000007; SubObjectsOfflineInfo.Highest sub-index supported.MinValue = '0x02'; SubObjectsOfflineInfo.Highest sub-index supported.MaxValue = '0x06'; SubObjectsOfflineInfo.Highest sub-index supported.AccessType = 'const'; SubObjectsOfflineInfo.Highest sub-index supported.IEC Variable = ''; SubObjectsOfflineInfo.Highest sub-index supported.DefaultValue = '0x5'; SubObjectsOfflineInfo.Highest sub-index supported.ObjectFlags = 16#00000000; SubObjectsOfflineInfo.COB-ID used by TPDO.Index = 16#00001801; SubObjectsOfflineInfo.COB-ID used by TPDO.SubIndex = 16#01; SubObjectsOfflineInfo.COB-ID used by TPDO.PDOMapping = FALSE; SubObjectsOfflineInfo.COB-ID used by TPDO.ObjectOwner = 16#03; SubObjectsOfflineInfo.COB-ID used by TPDO.ObjectType = 16#00000007; SubObjectsOfflineInfo.COB-ID used by TPDO.MinValue = '0x00000080'; SubObjectsOfflineInfo.COB-ID used by TPDO.MaxValue = '0xFFFFFFFF'; SubObjectsOfflineInfo.COB-ID used by TPDO.AccessType = 'rw';
            SubObjectsOfflineInfo.COB-ID used by TPDO.IEC Variable = ''; SubObjectsOfflineInfo.COB-ID used by TPDO.DefaultValue = '$$NODEID+0x280'; SubObjectsOfflineInfo.COB-ID used by TPDO.ObjectFlags = 16#00000000; SubObjectsOfflineInfo.Transmission type.Index = 16#00001801; SubObjectsOfflineInfo.Transmission type.SubIndex = 16#02; SubObjectsOfflineInfo.Transmission type.PDOMapping = FALSE; SubObjectsOfflineInfo.Transmission type.ObjectOwner = 16#03; SubObjectsOfflineInfo.Transmission type.ObjectType = 16#00000007; SubObjectsOfflineInfo.Transmission type.MinValue = '0x00'; SubObjectsOfflineInfo.Transmission type.MaxValue = '0xFF'; SubObjectsOfflineInfo.Transmission type.AccessType = 'rw'; SubObjectsOfflineInfo.Transmission type.IEC Variable = ''; SubObjectsOfflineInfo.Transmission type.DefaultValue = '0xFF'; SubObjectsOfflineInfo.Transmission type.ObjectFlags = 16#00000000; SubObjectsOfflineInfo.Inhibit time.Index = 16#00001801; SubObjectsOfflineInfo.Inhibit time.SubIndex = 16#03; SubObjectsOfflineInfo.Inhibit time.PDOMapping = FALSE; SubObjectsOfflineInfo.Inhibit time.ObjectOwner = 16#03; SubObjectsOfflineInfo.Inhibit time.ObjectType = 16#00000007; SubObjectsOfflineInfo.Inhibit time.MinValue = ''; SubObjectsOfflineInfo.Inhibit time.MaxValue = ''; SubObjectsOfflineInfo.Inhibit time.AccessType = 'rw'; SubObjectsOfflineInfo.Inhibit time.IEC Variable = ''; SubObjectsOfflineInfo.Inhibit time.DefaultValue = '0x0'; SubObjectsOfflineInfo.Inhibit time.ObjectFlags = 16#00000000; SubObjectsOfflineInfo.compatibility entry.Index = 16#00001801; SubObjectsOfflineInfo.compatibility entry.SubIndex = 16#04; SubObjectsOfflineInfo.compatibility entry.PDOMapping = FALSE; SubObjectsOfflineInfo.compatibility entry.ObjectOwner = 16#03; SubObjectsOfflineInfo.compatibility entry.ObjectType = 16#00000007; SubObjectsOfflineInfo.compatibility entry.MinValue = ''; SubObjectsOfflineInfo.compatibility entry.MaxValue = ''; SubObjectsOfflineInfo.compatibility entry.AccessType = 'rw'; SubObjectsOfflineInfo.compatibility entry.IEC Variable = ''; SubObjectsOfflineInfo.compatibility entry.DefaultValue = '0x0'; SubObjectsOfflineInfo.compatibility entry.ObjectFlags = 16#00000000; SubObjectsOfflineInfo.Event timer.Index = 16#00001801; SubObjectsOfflineInfo.Event timer.SubIndex = 16#05; SubObjectsOfflineInfo.Event timer.PDOMapping = FALSE; SubObjectsOfflineInfo.Event timer.ObjectOwner = 16#03;
            SubObjectsOfflineInfo.Event timer.ObjectType = 16#00000007; SubObjectsOfflineInfo.Event timer.MinValue = ''; SubObjectsOfflineInfo.Event timer.MaxValue = ''; SubObjectsOfflineInfo.Event timer.AccessType = 'rw'; SubObjectsOfflineInfo.Event timer.IEC Variable = ''; SubObjectsOfflineInfo.Event timer.DefaultValue = '0x0'; SubObjectsOfflineInfo.Event timer.ObjectFlags = 16#00000000; SubObjectsOfflineInfo.Highest sub-index supported.Index = 16#00001802; SubObjectsOfflineInfo.Highest sub-index supported.SubIndex = 16#00; SubObjectsOfflineInfo.Highest sub-index supported.PDOMapping = FALSE; SubObjectsOfflineInfo.Highest sub-index supported.ObjectOwner = 16#03; SubObjectsOfflineInfo.Highest sub-index supported.ObjectType = 16#00000007; SubObjectsOfflineInfo.Highest sub-index supported.MinValue = '0x02'; SubObjectsOfflineInfo.Highest sub-index supported.MaxValue = '0x06'; SubObjectsOfflineInfo.Highest sub-index supported.AccessType = 'const'; SubObjectsOfflineInfo.Highest sub-index supported.IEC Variable = ''; SubObjectsOfflineInfo.Highest sub-index supported.DefaultValue = '0x5'; SubObjectsOfflineInfo.Highest sub-index supported.ObjectFlags = 16#00000000; SubObjectsOfflineInfo.COB-ID used by TPDO.Index = 16#00001802; SubObjectsOfflineInfo.COB-ID used by TPDO.SubIndex = 16#01; SubObjectsOfflineInfo.COB-ID used by TPDO.PDOMapping = FALSE; SubObjectsOfflineInfo.COB-ID used by TPDO.ObjectOwner = 16#03; SubObjectsOfflineInfo.COB-ID used by TPDO.ObjectType = 16#00000007; SubObjectsOfflineInfo.COB-ID used by TPDO.MinValue = '0x00000080'; SubObjectsOfflineInfo.COB-ID used by TPDO.MaxValue = '0xFFFFFFFF'; SubObjectsOfflineInfo.COB-ID used by TPDO.AccessType = 'rw'; SubObjectsOfflineInfo.COB-ID used by TPDO.IEC Variable = ''; SubObjectsOfflineInfo.COB-ID used by TPDO.DefaultValue = '$$NODEID+0x380'; SubObjectsOfflineInfo.COB-ID used by TPDO.ObjectFlags = 16#00000000; SubObjectsOfflineInfo.Transmission type.Index = 16#00001802; SubObjectsOfflineInfo.Transmission type.SubIndex = 16#02; SubObjectsOfflineInfo.Transmission type.PDOMapping = FALSE; SubObjectsOfflineInfo.Transmission type.ObjectOwner = 16#03; SubObjectsOfflineInfo.Transmission type.ObjectType = 16#00000007; SubObjectsOfflineInfo.Transmission type.MinValue = '0x00'; SubObjectsOfflineInfo.Transmission type.MaxValue = '0xFF'; SubObjectsOfflineInfo.Transmission type.AccessType = 'rw'; SubObjectsOfflineInfo.Transmission type.IEC Variable = ''; SubObjectsOfflineInfo.Transmission type.DefaultValue = '0xFF'; SubObjectsOfflineInfo.Transmission type.ObjectFlags = 16#00000000;
            SubObjectsOfflineInfo.Inhibit time.Index = 16#00001802; SubObjectsOfflineInfo.Inhibit time.SubIndex = 16#03; SubObjectsOfflineInfo.Inhibit time.PDOMapping = FALSE; SubObjectsOfflineInfo.Inhibit time.ObjectOwner = 16#03; SubObjectsOfflineInfo.Inhibit time.ObjectType = 16#00000007; SubObjectsOfflineInfo.Inhibit time.MinValue = ''; SubObjectsOfflineInfo.Inhibit time.MaxValue = ''; SubObjectsOfflineInfo.Inhibit time.AccessType = 'rw'; SubObjectsOfflineInfo.Inhibit time.IEC Variable = ''; SubObjectsOfflineInfo.Inhibit time.DefaultValue = '0x0'; SubObjectsOfflineInfo.Inhibit time.ObjectFlags = 16#00000000; SubObjectsOfflineInfo.compatibility entry.Index = 16#00001802; SubObjectsOfflineInfo.compatibility entry.SubIndex = 16#04; SubObjectsOfflineInfo.compatibility entry.PDOMapping = FALSE; SubObjectsOfflineInfo.compatibility entry.ObjectOwner = 16#03; SubObjectsOfflineInfo.compatibility entry.ObjectType = 16#00000007; SubObjectsOfflineInfo.compatibility entry.MinValue = ''; SubObjectsOfflineInfo.compatibility entry.MaxValue = ''; SubObjectsOfflineInfo.compatibility entry.AccessType = 'rw'; SubObjectsOfflineInfo.compatibility entry.IEC Variable = ''; SubObjectsOfflineInfo.compatibility entry.DefaultValue = '0x0'; SubObjectsOfflineInfo.compatibility entry.ObjectFlags = 16#00000000; SubObjectsOfflineInfo.Event timer.Index = 16#00001802; SubObjectsOfflineInfo.Event timer.SubIndex = 16#05; SubObjectsOfflineInfo.Event timer.PDOMapping = FALSE; SubObjectsOfflineInfo.Event timer.ObjectOwner = 16#03; SubObjectsOfflineInfo.Event timer.ObjectType = 16#00000007; SubObjectsOfflineInfo.Event timer.MinValue = ''; SubObjectsOfflineInfo.Event timer.MaxValue = ''; SubObjectsOfflineInfo.Event timer.AccessType = 'rw'; SubObjectsOfflineInfo.Event timer.IEC Variable = ''; SubObjectsOfflineInfo.Event timer.DefaultValue = '0x0'; SubObjectsOfflineInfo.Event timer.ObjectFlags = 16#00000000; SubObjectsOfflineInfo.Number of mapped application objects in TPDO.Index = 16#00001A00; SubObjectsOfflineInfo.Number of mapped application objects in TPDO.SubIndex = 16#00; SubObjectsOfflineInfo.Number of mapped application objects in TPDO.PDOMapping = FALSE; SubObjectsOfflineInfo.Number of mapped application objects in TPDO.ObjectOwner = 16#03; SubObjectsOfflineInfo.Number of mapped application objects in TPDO.ObjectType = 16#00000007; SubObjectsOfflineInfo.Number of mapped application objects in TPDO.MinValue = '0'; SubObjectsOfflineInfo.Number of mapped application objects in TPDO.MaxValue = '8';
            SubObjectsOfflineInfo.Number of mapped application objects in TPDO.AccessType = 'const'; SubObjectsOfflineInfo.Number of mapped application objects in TPDO.IEC Variable = ''; SubObjectsOfflineInfo.Number of mapped application objects in TPDO.DefaultValue = '0x04'; SubObjectsOfflineInfo.Number of mapped application objects in TPDO.ObjectFlags = 16#00000000; SubObjectsOfflineInfo.Mapping Entry.Index = 16#00001A00; SubObjectsOfflineInfo.Mapping Entry.SubIndex = 16#01; SubObjectsOfflineInfo.Mapping Entry.PDOMapping = FALSE; SubObjectsOfflineInfo.Mapping Entry.ObjectOwner = 16#03; SubObjectsOfflineInfo.Mapping Entry.ObjectType = 16#00000007; SubObjectsOfflineInfo.Mapping Entry.MinValue = '0x0'; SubObjectsOfflineInfo.Mapping Entry.MaxValue = '0xFFFFFFFF'; SubObjectsOfflineInfo.Mapping Entry.AccessType = 'const'; SubObjectsOfflineInfo.Mapping Entry.IEC Variable = ''; SubObjectsOfflineInfo.Mapping Entry.DefaultValue = '0x38000110'; SubObjectsOfflineInfo.Mapping Entry.ObjectFlags = 16#00000000; SubObjectsOfflineInfo.Mapping Entry.Index = 16#00001A00; SubObjectsOfflineInfo.Mapping Entry.SubIndex = 16#02; SubObjectsOfflineInfo.Mapping Entry.PDOMapping = FALSE; SubObjectsOfflineInfo.Mapping Entry.ObjectOwner = 16#03; SubObjectsOfflineInfo.Mapping Entry.ObjectType = 16#00000007; SubObjectsOfflineInfo.Mapping Entry.MinValue = '0x0'; SubObjectsOfflineInfo.Mapping Entry.MaxValue = '0xFFFFFFFF'; SubObjectsOfflineInfo.Mapping Entry.AccessType = 'const'; SubObjectsOfflineInfo.Mapping Entry.IEC Variable = ''; SubObjectsOfflineInfo.Mapping Entry.DefaultValue = '0x38010110'; SubObjectsOfflineInfo.Mapping Entry.ObjectFlags = 16#00000000; SubObjectsOfflineInfo.Mapping Entry.Index = 16#00001A00; SubObjectsOfflineInfo.Mapping Entry.SubIndex = 16#03; SubObjectsOfflineInfo.Mapping Entry.PDOMapping = FALSE; SubObjectsOfflineInfo.Mapping Entry.ObjectOwner = 16#03; SubObjectsOfflineInfo.Mapping Entry.ObjectType = 16#00000007; SubObjectsOfflineInfo.Mapping Entry.MinValue = '0x0'; SubObjectsOfflineInfo.Mapping Entry.MaxValue = '0xFFFFFFFF'; SubObjectsOfflineInfo.Mapping Entry.AccessType = 'const'; SubObjectsOfflineInfo.Mapping Entry.IEC Variable = ''; SubObjectsOfflineInfo.Mapping Entry.DefaultValue = '0x38020108'; SubObjectsOfflineInfo.Mapping Entry.ObjectFlags = 16#00000000; SubObjectsOfflineInfo.Mapping Entry.Index = 16#00001A00; SubObjectsOfflineInfo.Mapping Entry.SubIndex = 16#04; SubObjectsOfflineInfo.Mapping Entry.PDOMapping = FALSE;
            SubObjectsOfflineInfo.Mapping Entry.ObjectOwner = 16#03; SubObjectsOfflineInfo.Mapping Entry.ObjectType = 16#00000007; SubObjectsOfflineInfo.Mapping Entry.MinValue = '0x0'; SubObjectsOfflineInfo.Mapping Entry.MaxValue = '0xFFFFFFFF'; SubObjectsOfflineInfo.Mapping Entry.AccessType = 'const'; SubObjectsOfflineInfo.Mapping Entry.IEC Variable = ''; SubObjectsOfflineInfo.Mapping Entry.DefaultValue = '0x38030108'; SubObjectsOfflineInfo.Mapping Entry.ObjectFlags = 16#00000000; SubObjectsOfflineInfo.Number of mapped application objects in TPDO.Index = 16#00001A01; SubObjectsOfflineInfo.Number of mapped application objects in TPDO.SubIndex = 16#00; SubObjectsOfflineInfo.Number of mapped application objects in TPDO.PDOMapping = FALSE; SubObjectsOfflineInfo.Number of mapped application objects in TPDO.ObjectOwner = 16#03; SubObjectsOfflineInfo.Number of mapped application objects in TPDO.ObjectType = 16#00000007; SubObjectsOfflineInfo.Number of mapped application objects in TPDO.MinValue = '0'; SubObjectsOfflineInfo.Number of mapped application objects in TPDO.MaxValue = '8'; SubObjectsOfflineInfo.Number of mapped application objects in TPDO.AccessType = 'const'; SubObjectsOfflineInfo.Number of mapped application objects in TPDO.IEC Variable = ''; SubObjectsOfflineInfo.Number of mapped application objects in TPDO.DefaultValue = '0x02'; SubObjectsOfflineInfo.Number of mapped application objects in TPDO.ObjectFlags = 16#00000000; SubObjectsOfflineInfo.Mapping Entry.Index = 16#00001A01; SubObjectsOfflineInfo.Mapping Entry.SubIndex = 16#01; SubObjectsOfflineInfo.Mapping Entry.PDOMapping = FALSE; SubObjectsOfflineInfo.Mapping Entry.ObjectOwner = 16#03; SubObjectsOfflineInfo.Mapping Entry.ObjectType = 16#00000007; SubObjectsOfflineInfo.Mapping Entry.MinValue = '0x0'; SubObjectsOfflineInfo.Mapping Entry.MaxValue = '0xFFFFFFFF'; SubObjectsOfflineInfo.Mapping Entry.AccessType = 'const'; SubObjectsOfflineInfo.Mapping Entry.IEC Variable = ''; SubObjectsOfflineInfo.Mapping Entry.DefaultValue = '0x38040120'; SubObjectsOfflineInfo.Mapping Entry.ObjectFlags = 16#00000000; SubObjectsOfflineInfo.Mapping Entry.Index = 16#00001A01; SubObjectsOfflineInfo.Mapping Entry.SubIndex = 16#02; SubObjectsOfflineInfo.Mapping Entry.PDOMapping = FALSE; SubObjectsOfflineInfo.Mapping Entry.ObjectOwner = 16#03; SubObjectsOfflineInfo.Mapping Entry.ObjectType = 16#00000007; SubObjectsOfflineInfo.Mapping Entry.MinValue = '0x0'; SubObjectsOfflineInfo.Mapping Entry.MaxValue = '0xFFFFFFFF'; SubObjectsOfflineInfo.Mapping Entry.AccessType = 'const'; SubObjectsOfflineInfo.Mapping Entry.IEC Variable = ''; SubObjectsOfflineInfo.Mapping Entry.DefaultValue = '0x38050110';
            SubObjectsOfflineInfo.Mapping Entry.ObjectFlags = 16#00000000; SubObjectsOfflineInfo.Number of mapped application objects in TPDO.Index = 16#00001A02; SubObjectsOfflineInfo.Number of mapped application objects in TPDO.SubIndex = 16#00; SubObjectsOfflineInfo.Number of mapped application objects in TPDO.PDOMapping = FALSE; SubObjectsOfflineInfo.Number of mapped application objects in TPDO.ObjectOwner = 16#03; SubObjectsOfflineInfo.Number of mapped application objects in TPDO.ObjectType = 16#00000007; SubObjectsOfflineInfo.Number of mapped application objects in TPDO.MinValue = '0'; SubObjectsOfflineInfo.Number of mapped application objects in TPDO.MaxValue = '8'; SubObjectsOfflineInfo.Number of mapped application objects in TPDO.AccessType = 'const'; SubObjectsOfflineInfo.Number of mapped application objects in TPDO.IEC Variable = ''; SubObjectsOfflineInfo.Number of mapped application objects in TPDO.DefaultValue = '0x03'; SubObjectsOfflineInfo.Number of mapped application objects in TPDO.ObjectFlags = 16#00000000; SubObjectsOfflineInfo.Mapping Entry.Index = 16#00001A02; SubObjectsOfflineInfo.Mapping Entry.SubIndex = 16#01; SubObjectsOfflineInfo.Mapping Entry.PDOMapping = FALSE; SubObjectsOfflineInfo.Mapping Entry.ObjectOwner = 16#03; SubObjectsOfflineInfo.Mapping Entry.ObjectType = 16#00000007; SubObjectsOfflineInfo.Mapping Entry.MinValue = '0x0'; SubObjectsOfflineInfo.Mapping Entry.MaxValue = '0xFFFFFFFF'; SubObjectsOfflineInfo.Mapping Entry.AccessType = 'const'; SubObjectsOfflineInfo.Mapping Entry.IEC Variable = ''; SubObjectsOfflineInfo.Mapping Entry.DefaultValue = '0x38060110'; SubObjectsOfflineInfo.Mapping Entry.ObjectFlags = 16#00000000; SubObjectsOfflineInfo.Mapping Entry.Index = 16#00001A02; SubObjectsOfflineInfo.Mapping Entry.SubIndex = 16#02; SubObjectsOfflineInfo.Mapping Entry.PDOMapping = FALSE; SubObjectsOfflineInfo.Mapping Entry.ObjectOwner = 16#03; SubObjectsOfflineInfo.Mapping Entry.ObjectType = 16#00000007; SubObjectsOfflineInfo.Mapping Entry.MinValue = '0x0'; SubObjectsOfflineInfo.Mapping Entry.MaxValue = '0xFFFFFFFF'; SubObjectsOfflineInfo.Mapping Entry.AccessType = 'const'; SubObjectsOfflineInfo.Mapping Entry.IEC Variable = ''; SubObjectsOfflineInfo.Mapping Entry.DefaultValue = '0x38060210'; SubObjectsOfflineInfo.Mapping Entry.ObjectFlags = 16#00000000; SubObjectsOfflineInfo.Mapping Entry.Index = 16#00001A02; SubObjectsOfflineInfo.Mapping Entry.SubIndex = 16#03; SubObjectsOfflineInfo.Mapping Entry.PDOMapping = FALSE; SubObjectsOfflineInfo.Mapping Entry.ObjectOwner = 16#03; SubObjectsOfflineInfo.Mapping Entry.ObjectType = 16#00000007; SubObjectsOfflineInfo.Mapping Entry.MinValue = '0x0';
            SubObjectsOfflineInfo.Mapping Entry.MaxValue = '0xFFFFFFFF'; SubObjectsOfflineInfo.Mapping Entry.AccessType = 'const'; SubObjectsOfflineInfo.Mapping Entry.IEC Variable = ''; SubObjectsOfflineInfo.Mapping Entry.DefaultValue = '0x38060310'; SubObjectsOfflineInfo.Mapping Entry.ObjectFlags = 16#00000000; SubObjectsOfflineInfo.Number of Entries.Index = 16#00003000; SubObjectsOfflineInfo.Number of Entries.SubIndex = 16#00; SubObjectsOfflineInfo.Number of Entries.PDOMapping = FALSE; SubObjectsOfflineInfo.Number of Entries.ObjectOwner = 16#03; SubObjectsOfflineInfo.Number of Entries.ObjectType = 16#00000007; SubObjectsOfflineInfo.Number of Entries.MinValue = ''; SubObjectsOfflineInfo.Number of Entries.MaxValue = ''; SubObjectsOfflineInfo.Number of Entries.AccessType = 'const'; SubObjectsOfflineInfo.Number of Entries.IEC Variable = ''; SubObjectsOfflineInfo.Number of Entries.DefaultValue = '0x01'; SubObjectsOfflineInfo.Number of Entries.ObjectFlags = 16#00000000; SubObjectsOfflineInfo.set_speed.Index = 16#00003000; SubObjectsOfflineInfo.set_speed.SubIndex = 16#01; SubObjectsOfflineInfo.set_speed.PDOMapping = TRUE; SubObjectsOfflineInfo.set_speed.ObjectOwner = 16#03; SubObjectsOfflineInfo.set_speed.ObjectType = 16#00000007; SubObjectsOfflineInfo.set_speed.MinValue = ''; SubObjectsOfflineInfo.set_speed.MaxValue = ''; SubObjectsOfflineInfo.set_speed.AccessType = 'rww'; SubObjectsOfflineInfo.set_speed.IEC Variable = ''; SubObjectsOfflineInfo.set_speed.DefaultValue = ''; SubObjectsOfflineInfo.set_speed.ObjectFlags = 16#00000000; SubObjectsOfflineInfo.Number of Entries.Index = 16#00003001; SubObjectsOfflineInfo.Number of Entries.SubIndex = 16#00; SubObjectsOfflineInfo.Number of Entries.PDOMapping = FALSE; SubObjectsOfflineInfo.Number of Entries.ObjectOwner = 16#03; SubObjectsOfflineInfo.Number of Entries.ObjectType = 16#00000007; SubObjectsOfflineInfo.Number of Entries.MinValue = ''; SubObjectsOfflineInfo.Number of Entries.MaxValue = ''; SubObjectsOfflineInfo.Number of Entries.AccessType = 'const'; SubObjectsOfflineInfo.Number of Entries.IEC Variable = ''; SubObjectsOfflineInfo.Number of Entries.DefaultValue = '0x01'; SubObjectsOfflineInfo.Number of Entries.ObjectFlags = 16#00000000; SubObjectsOfflineInfo.set_acc_time.Index = 16#00003001; SubObjectsOfflineInfo.set_acc_time.SubIndex = 16#01;
            SubObjectsOfflineInfo.set_acc_time.PDOMapping = TRUE; SubObjectsOfflineInfo.set_acc_time.ObjectOwner = 16#03; SubObjectsOfflineInfo.set_acc_time.ObjectType = 16#00000007; SubObjectsOfflineInfo.set_acc_time.MinValue = ''; SubObjectsOfflineInfo.set_acc_time.MaxValue = ''; SubObjectsOfflineInfo.set_acc_time.AccessType = 'rww'; SubObjectsOfflineInfo.set_acc_time.IEC Variable = ''; SubObjectsOfflineInfo.set_acc_time.DefaultValue = ''; SubObjectsOfflineInfo.set_acc_time.ObjectFlags = 16#00000000; SubObjectsOfflineInfo.Number of Entries.Index = 16#00003002; SubObjectsOfflineInfo.Number of Entries.SubIndex = 16#00; SubObjectsOfflineInfo.Number of Entries.PDOMapping = FALSE; SubObjectsOfflineInfo.Number of Entries.ObjectOwner = 16#03; SubObjectsOfflineInfo.Number of Entries.ObjectType = 16#00000007; SubObjectsOfflineInfo.Number of Entries.MinValue = ''; SubObjectsOfflineInfo.Number of Entries.MaxValue = ''; SubObjectsOfflineInfo.Number of Entries.AccessType = 'const'; SubObjectsOfflineInfo.Number of Entries.IEC Variable = ''; SubObjectsOfflineInfo.Number of Entries.DefaultValue = '0x01'; SubObjectsOfflineInfo.Number of Entries.ObjectFlags = 16#00000000; SubObjectsOfflineInfo.set_current_limit.Index = 16#00003002; SubObjectsOfflineInfo.set_current_limit.SubIndex = 16#01; SubObjectsOfflineInfo.set_current_limit.PDOMapping = TRUE; SubObjectsOfflineInfo.set_current_limit.ObjectOwner = 16#03; SubObjectsOfflineInfo.set_current_limit.ObjectType = 16#00000007; SubObjectsOfflineInfo.set_current_limit.MinValue = ''; SubObjectsOfflineInfo.set_current_limit.MaxValue = ''; SubObjectsOfflineInfo.set_current_limit.AccessType = 'rww'; SubObjectsOfflineInfo.set_current_limit.IEC Variable = ''; SubObjectsOfflineInfo.set_current_limit.DefaultValue = ''; SubObjectsOfflineInfo.set_current_limit.ObjectFlags = 16#00000000; SubObjectsOfflineInfo.Number of Entries.Index = 16#00003003; SubObjectsOfflineInfo.Number of Entries.SubIndex = 16#00; SubObjectsOfflineInfo.Number of Entries.PDOMapping = FALSE; SubObjectsOfflineInfo.Number of Entries.ObjectOwner = 16#03; SubObjectsOfflineInfo.Number of Entries.ObjectType = 16#00000007; SubObjectsOfflineInfo.Number of Entries.MinValue = ''; SubObjectsOfflineInfo.Number of Entries.MaxValue = ''; SubObjectsOfflineInfo.Number of Entries.AccessType = 'const'; SubObjectsOfflineInfo.Number of Entries.IEC Variable = '';
            SubObjectsOfflineInfo.Number of Entries.DefaultValue = '0x01'; SubObjectsOfflineInfo.Number of Entries.ObjectFlags = 16#00000000; SubObjectsOfflineInfo.set_cmd.Index = 16#00003003; SubObjectsOfflineInfo.set_cmd.SubIndex = 16#01; SubObjectsOfflineInfo.set_cmd.PDOMapping = TRUE; SubObjectsOfflineInfo.set_cmd.ObjectOwner = 16#03; SubObjectsOfflineInfo.set_cmd.ObjectType = 16#00000007; SubObjectsOfflineInfo.set_cmd.MinValue = ''; SubObjectsOfflineInfo.set_cmd.MaxValue = ''; SubObjectsOfflineInfo.set_cmd.AccessType = 'rww'; SubObjectsOfflineInfo.set_cmd.IEC Variable = ''; SubObjectsOfflineInfo.set_cmd.DefaultValue = ''; SubObjectsOfflineInfo.set_cmd.ObjectFlags = 16#00000000; SubObjectsOfflineInfo.Number of Entries.Index = 16#00003800; SubObjectsOfflineInfo.Number of Entries.SubIndex = 16#00; SubObjectsOfflineInfo.Number of Entries.PDOMapping = FALSE; SubObjectsOfflineInfo.Number of Entries.ObjectOwner = 16#03; SubObjectsOfflineInfo.Number of Entries.ObjectType = 16#00000007; SubObjectsOfflineInfo.Number of Entries.MinValue = ''; SubObjectsOfflineInfo.Number of Entries.MaxValue = ''; SubObjectsOfflineInfo.Number of Entries.AccessType = 'const'; SubObjectsOfflineInfo.Number of Entries.IEC Variable = ''; SubObjectsOfflineInfo.Number of Entries.DefaultValue = '0x01'; SubObjectsOfflineInfo.Number of Entries.ObjectFlags = 16#00000000; SubObjectsOfflineInfo.speed.Index = 16#00003800; SubObjectsOfflineInfo.speed.SubIndex = 16#01; SubObjectsOfflineInfo.speed.PDOMapping = TRUE; SubObjectsOfflineInfo.speed.ObjectOwner = 16#03; SubObjectsOfflineInfo.speed.ObjectType = 16#00000007; SubObjectsOfflineInfo.speed.MinValue = ''; SubObjectsOfflineInfo.speed.MaxValue = ''; SubObjectsOfflineInfo.speed.AccessType = 'ro'; SubObjectsOfflineInfo.speed.IEC Variable = ''; SubObjectsOfflineInfo.speed.DefaultValue = ''; SubObjectsOfflineInfo.speed.ObjectFlags = 16#00000000; SubObjectsOfflineInfo.Number of Entries.Index = 16#00003801; SubObjectsOfflineInfo.Number of Entries.SubIndex = 16#00; SubObjectsOfflineInfo.Number of Entries.PDOMapping = FALSE; SubObjectsOfflineInfo.Number of Entries.ObjectOwner = 16#03; SubObjectsOfflineInfo.Number of Entries.ObjectType = 16#00000007;
            SubObjectsOfflineInfo.Number of Entries.MinValue = ''; SubObjectsOfflineInfo.Number of Entries.MaxValue = ''; SubObjectsOfflineInfo.Number of Entries.AccessType = 'const'; SubObjectsOfflineInfo.Number of Entries.IEC Variable = ''; SubObjectsOfflineInfo.Number of Entries.DefaultValue = '0x01'; SubObjectsOfflineInfo.Number of Entries.ObjectFlags = 16#00000000; SubObjectsOfflineInfo.current.Index = 16#00003801; SubObjectsOfflineInfo.current.SubIndex = 16#01; SubObjectsOfflineInfo.current.PDOMapping = TRUE; SubObjectsOfflineInfo.current.ObjectOwner = 16#03; SubObjectsOfflineInfo.current.ObjectType = 16#00000007; SubObjectsOfflineInfo.current.MinValue = ''; SubObjectsOfflineInfo.current.MaxValue = ''; SubObjectsOfflineInfo.current.AccessType = 'ro'; SubObjectsOfflineInfo.current.IEC Variable = ''; SubObjectsOfflineInfo.current.DefaultValue = ''; SubObjectsOfflineInfo.current.ObjectFlags = 16#00000000; SubObjectsOfflineInfo.Number of Entries.Index = 16#00003802; SubObjectsOfflineInfo.Number of Entries.SubIndex = 16#00; SubObjectsOfflineInfo.Number of Entries.PDOMapping = FALSE; SubObjectsOfflineInfo.Number of Entries.ObjectOwner = 16#03; SubObjectsOfflineInfo.Number of Entries.ObjectType = 16#00000007; SubObjectsOfflineInfo.Number of Entries.MinValue = ''; SubObjectsOfflineInfo.Number of Entries.MaxValue = ''; SubObjectsOfflineInfo.Number of Entries.AccessType = 'const'; SubObjectsOfflineInfo.Number of Entries.IEC Variable = ''; SubObjectsOfflineInfo.Number of Entries.DefaultValue = '0x01'; SubObjectsOfflineInfo.Number of Entries.ObjectFlags = 16#00000000; SubObjectsOfflineInfo.acc_time.Index = 16#00003802; SubObjectsOfflineInfo.acc_time.SubIndex = 16#01; SubObjectsOfflineInfo.acc_time.PDOMapping = TRUE; SubObjectsOfflineInfo.acc_time.ObjectOwner = 16#03; SubObjectsOfflineInfo.acc_time.ObjectType = 16#00000007; SubObjectsOfflineInfo.acc_time.MinValue = ''; SubObjectsOfflineInfo.acc_time.MaxValue = ''; SubObjectsOfflineInfo.acc_time.AccessType = 'ro'; SubObjectsOfflineInfo.acc_time.IEC Variable = ''; SubObjectsOfflineInfo.acc_time.DefaultValue = ''; SubObjectsOfflineInfo.acc_time.ObjectFlags = 16#00000000; SubObjectsOfflineInfo.Number of Entries.Index = 16#00003803;
            SubObjectsOfflineInfo.Number of Entries.SubIndex = 16#00; SubObjectsOfflineInfo.Number of Entries.PDOMapping = FALSE; SubObjectsOfflineInfo.Number of Entries.ObjectOwner = 16#03; SubObjectsOfflineInfo.Number of Entries.ObjectType = 16#00000007; SubObjectsOfflineInfo.Number of Entries.MinValue = ''; SubObjectsOfflineInfo.Number of Entries.MaxValue = ''; SubObjectsOfflineInfo.Number of Entries.AccessType = 'const'; SubObjectsOfflineInfo.Number of Entries.IEC Variable = ''; SubObjectsOfflineInfo.Number of Entries.DefaultValue = '0x01'; SubObjectsOfflineInfo.Number of Entries.ObjectFlags = 16#00000000; SubObjectsOfflineInfo.temperature.Index = 16#00003803; SubObjectsOfflineInfo.temperature.SubIndex = 16#01; SubObjectsOfflineInfo.temperature.PDOMapping = TRUE; SubObjectsOfflineInfo.temperature.ObjectOwner = 16#03; SubObjectsOfflineInfo.temperature.ObjectType = 16#00000007; SubObjectsOfflineInfo.temperature.MinValue = ''; SubObjectsOfflineInfo.temperature.MaxValue = ''; SubObjectsOfflineInfo.temperature.AccessType = 'ro'; SubObjectsOfflineInfo.temperature.IEC Variable = ''; SubObjectsOfflineInfo.temperature.DefaultValue = ''; SubObjectsOfflineInfo.temperature.ObjectFlags = 16#00000000; SubObjectsOfflineInfo.Number of Entries.Index = 16#00003804; SubObjectsOfflineInfo.Number of Entries.SubIndex = 16#00; SubObjectsOfflineInfo.Number of Entries.PDOMapping = FALSE; SubObjectsOfflineInfo.Number of Entries.ObjectOwner = 16#03; SubObjectsOfflineInfo.Number of Entries.ObjectType = 16#00000007; SubObjectsOfflineInfo.Number of Entries.MinValue = ''; SubObjectsOfflineInfo.Number of Entries.MaxValue = ''; SubObjectsOfflineInfo.Number of Entries.AccessType = 'const'; SubObjectsOfflineInfo.Number of Entries.IEC Variable = ''; SubObjectsOfflineInfo.Number of Entries.DefaultValue = '0x01'; SubObjectsOfflineInfo.Number of Entries.ObjectFlags = 16#00000000; SubObjectsOfflineInfo.dummy.Index = 16#00003804; SubObjectsOfflineInfo.dummy.SubIndex = 16#01; SubObjectsOfflineInfo.dummy.PDOMapping = TRUE; SubObjectsOfflineInfo.dummy.ObjectOwner = 16#03; SubObjectsOfflineInfo.dummy.ObjectType = 16#00000007; SubObjectsOfflineInfo.dummy.MinValue = ''; SubObjectsOfflineInfo.dummy.MaxValue = ''; SubObjectsOfflineInfo.dummy.AccessType = 'ro';
            SubObjectsOfflineInfo.dummy.IEC Variable = ''; SubObjectsOfflineInfo.dummy.DefaultValue = ''; SubObjectsOfflineInfo.dummy.ObjectFlags = 16#00000000; SubObjectsOfflineInfo.Number of Entries.Index = 16#00003805; SubObjectsOfflineInfo.Number of Entries.SubIndex = 16#00; SubObjectsOfflineInfo.Number of Entries.PDOMapping = FALSE; SubObjectsOfflineInfo.Number of Entries.ObjectOwner = 16#03; SubObjectsOfflineInfo.Number of Entries.ObjectType = 16#00000007; SubObjectsOfflineInfo.Number of Entries.MinValue = ''; SubObjectsOfflineInfo.Number of Entries.MaxValue = ''; SubObjectsOfflineInfo.Number of Entries.AccessType = 'ro'; SubObjectsOfflineInfo.Number of Entries.IEC Variable = ''; SubObjectsOfflineInfo.Number of Entries.DefaultValue = '0x1'; SubObjectsOfflineInfo.Number of Entries.ObjectFlags = 16#00000000; SubObjectsOfflineInfo.error_code.Index = 16#00003805; SubObjectsOfflineInfo.error_code.SubIndex = 16#01; SubObjectsOfflineInfo.error_code.PDOMapping = TRUE; SubObjectsOfflineInfo.error_code.ObjectOwner = 16#03; SubObjectsOfflineInfo.error_code.ObjectType = 16#00000007; SubObjectsOfflineInfo.error_code.MinValue = ''; SubObjectsOfflineInfo.error_code.MaxValue = ''; SubObjectsOfflineInfo.error_code.AccessType = 'ro'; SubObjectsOfflineInfo.error_code.IEC Variable = ''; SubObjectsOfflineInfo.error_code.DefaultValue = ''; SubObjectsOfflineInfo.error_code.ObjectFlags = 16#00000000; SubObjectsOfflineInfo.Number of Entries.Index = 16#00003806; SubObjectsOfflineInfo.Number of Entries.SubIndex = 16#00; SubObjectsOfflineInfo.Number of Entries.PDOMapping = FALSE; SubObjectsOfflineInfo.Number of Entries.ObjectOwner = 16#03; SubObjectsOfflineInfo.Number of Entries.ObjectType = 16#00000007; SubObjectsOfflineInfo.Number of Entries.MinValue = ''; SubObjectsOfflineInfo.Number of Entries.MaxValue = ''; SubObjectsOfflineInfo.Number of Entries.AccessType = 'ro'; SubObjectsOfflineInfo.Number of Entries.IEC Variable = ''; SubObjectsOfflineInfo.Number of Entries.DefaultValue = '0x3'; SubObjectsOfflineInfo.Number of Entries.ObjectFlags = 16#00000000; SubObjectsOfflineInfo.yaw.Index = 16#00003806; SubObjectsOfflineInfo.yaw.SubIndex = 16#01; SubObjectsOfflineInfo.yaw.PDOMapping = TRUE; SubObjectsOfflineInfo.yaw.ObjectOwner = 16#03;
            SubObjectsOfflineInfo.yaw.ObjectType = 16#00000007; SubObjectsOfflineInfo.yaw.MinValue = ''; SubObjectsOfflineInfo.yaw.MaxValue = ''; SubObjectsOfflineInfo.yaw.AccessType = 'ro'; SubObjectsOfflineInfo.yaw.IEC Variable = ''; SubObjectsOfflineInfo.yaw.DefaultValue = ''; SubObjectsOfflineInfo.yaw.ObjectFlags = 16#00000000; SubObjectsOfflineInfo.pitch.Index = 16#00003806; SubObjectsOfflineInfo.pitch.SubIndex = 16#02; SubObjectsOfflineInfo.pitch.PDOMapping = TRUE; SubObjectsOfflineInfo.pitch.ObjectOwner = 16#03; SubObjectsOfflineInfo.pitch.ObjectType = 16#00000007; SubObjectsOfflineInfo.pitch.MinValue = ''; SubObjectsOfflineInfo.pitch.MaxValue = ''; SubObjectsOfflineInfo.pitch.AccessType = 'ro'; SubObjectsOfflineInfo.pitch.IEC Variable = ''; SubObjectsOfflineInfo.pitch.DefaultValue = ''; SubObjectsOfflineInfo.pitch.ObjectFlags = 16#00000000; SubObjectsOfflineInfo.roll.Index = 16#00003806; SubObjectsOfflineInfo.roll.SubIndex = 16#03; SubObjectsOfflineInfo.roll.PDOMapping = TRUE; SubObjectsOfflineInfo.roll.ObjectOwner = 16#03; SubObjectsOfflineInfo.roll.ObjectType = 16#00000007; SubObjectsOfflineInfo.roll.MinValue = ''; SubObjectsOfflineInfo.roll.MaxValue = ''; SubObjectsOfflineInfo.roll.AccessType = 'ro'; SubObjectsOfflineInfo.roll.IEC Variable = ''; SubObjectsOfflineInfo.roll.DefaultValue = ''; SubObjectsOfflineInfo.roll.ObjectFlags = 16#00000000
          unmapped channels: set_speed, set_acc_time, set_current_limit, set_cmd, speed, current, acc_time, temperature, dummy, error_code, yaw, pitch, roll
  libraries: VisuSymbols, 4.5.0.0 (System); DepictorBase, 1.2.0.0 (CODESYS)
  text list GlobalTextList
  5ce3da45-db07-42e7-a21c-a00fff4ed8f6|C:\Users\phe\Downloads\Musterloesung_FUP.PNG
*)

// xLH_base/app/MAIN
PROGRAM MAIN
VAR

END_VAR

END_PROGRAM
